(* PLC project common, CODESYS STW CODESYS V3.5 SP11 - ESX-3CS *)
(* stored: creationDateTime 2026-05-19T11:31:35.1210252, version 0.1, modificationDateTime 2026-01-27T11:29:48, organization Isoloader *)

TYPE t_can_message : CANMessage;
END_TYPE

TYPE t_can_message_set : ARRAY[1..32] OF POINTER TO t_can_message;
END_TYPE

TYPE t_long_string : STRING(72);
END_TYPE

TYPE t_long_string_reference : REFERENCE TO t_long_string;
END_TYPE

TYPE t_medium_string : STRING(16);
END_TYPE

TYPE t_medium_string_reference : REFERENCE TO t_medium_string;
END_TYPE

TYPE t_mediumlong_string : STRING(32);
END_TYPE

TYPE t_mediumlong_string_reference : REFERENCE TO t_mediumlong_string;
END_TYPE

TYPE t_ms_time : TIME;
END_TYPE

TYPE t_onoff_state : (cOnOffStateOff := 0, cOnOffStateTurningOn := 1, cOnOffStateOn := 2, cOnOffStateTurningOff := 3);
END_TYPE

TYPE t_percentage : REAL;
END_TYPE

TYPE t_short_string : STRING(8);
END_TYPE

TYPE t_short_string_reference : REFERENCE TO t_short_string;
END_TYPE

TYPE t_time : TIME;
END_TYPE

TYPE t_timer : Timer;
END_TYPE

TYPE t_system_handler : SystemHandler;
END_TYPE

VAR_GLOBAL CONSTANT  (* GlobalVariablesCommon *)
  cPi : REAL := 3.141592654;
  c2Pi : REAL := 6.283185307;
  cPiNegative : REAL := -3.141592654;
  cPIOn2 : REAL := 1.5708;
  cRelayCoilCurrentMinThreshold : WORD := 200;
  cRelayCoilCurrentMaxThreshold : WORD := 500;
  cRelayCoilResistanceThreshold : WORD := 80;
  cRelayCoilCurrentThreshold : WORD := 200;
  cRelayCoilTimeout : t_time := TIME#500ms;
  cRelayCoilTimeoutIndirect : t_time := TIME#600ms;
  gCodeErrorHandler : t_system_handler;
  gConfigErrorHandler : t_system_handler;
  gManualTemporaryOveride : BOOL := FALSE;
END_VAR

FUNCTION_BLOCK CANMessage
  VAR
    lSuccess : BOOL;
    lProceed : BOOL;
    lFinished : BOOL;
    lStarted : BOOL;
    lMessageCount : UINT := 0;
    lPostTimer : t_timer;
  END_VAR

            
          

METHOD finish
                  reset();

lStarted := TRUE;
lMessageCount := lMessageCount + 1;
                
END_METHOD

METHOD initialize
                  reset();

lMessageCount := 0;

lPostTimer.Enable := TRUE;
lPostTimer.Period := T#5S;
lPostTimer.initialize();
                
END_METHOD

METHOD operator
                  IF (NOT(Finished)) then
	lPostTimer.reset();
END_IF

lPostTimer.operator();

                
END_METHOD

METHOD reset
                  lSuccess := FALSE;
lProceed := FALSE;
lFinished := FALSE;
lStarted := FALSE;

                
END_METHOD

METHOD start
                  reset();

lStarted := TRUE;
lMessageCount := lMessageCount + 1;
                
END_METHOD

PROPERTY Finished : BOOL
GET
                    Finished := lFinished;
                  
END_GET
END_PROPERTY

PROPERTY PostPeriod : t_time
GET
                    PostPeriod := lPostTImer.Period;
                  
END_GET
SET
                    lPostTimer.Period := PostPeriod;
                  
END_SET
END_PROPERTY

PROPERTY Proceed : BOOL
GET
                    Proceed := lProceed;
                  
END_GET
END_PROPERTY

PROPERTY Running : BOOL
GET
                    Running := ((lStarted) and (NOT(lPostTimer.Expired)));
                  
END_GET
END_PROPERTY

PROPERTY Started : BOOL
GET
                    Started := lStarted;
                  
END_GET
END_PROPERTY

PROPERTY Success : BOOL
GET
                    Success := lSuccess;
                  
END_GET
END_PROPERTY
END_FUNCTION_BLOCK

FUNCTION_BLOCK CANMessageSequence EXTENDS CANMessage
  VAR
    lSequence : t_can_message_set;
    lSequenceCount : USINT := 0;
    lSequenceIndex : USINT := 0;
  END_VAR

            
          

METHOD initialize
  VAR
    i : USINT;
  END_VAR
                  SUPER^.initialize();

FOR i:=1 TO lSequenceCount DO
	lSequence[i]^.initialize();
END_FOR

                
END_METHOD

METHOD operator
  VAR
    b : BOOL;
  END_VAR
                  IF ((NOT(Enabled)) OR (NOT(Running))) THEN
	RETURN;
END_IF

SUPER^.operator();

lSequence[lSequenceIndex]^.operator();

IF (lSequence[lSequenceIndex]^.Finished) THEN
	IF (lSequence[lSequenceIndex]^.Proceed) THEN
		b:= lSequence[lSequenceIndex]^.Success;
		
		lSequenceIndex := lSequenceIndex + 1;
		IF (lSequenceIndex>lSequenceCount) THEN
			lSuccess := b;
			lFinished := TRUE;
			finish();
		ELSE
			lSequence[lSequenceIndex]^.start();	
		END_IF
	ELSE
		lSuccess := FALSE;
		lFinished := TRUE;
		finish();
	END_IF
END_IF

                
END_METHOD

METHOD registerMessage : POINTER TO t_can_message
  VAR_INPUT
    message : POINTER TO t_can_message;
  END_VAR
                  IF (lSequenceCount>32) THEN
	registerMessage := 0;
	RETURN;
END_IF

lSequenceCount := lSequenceCount + 1;
lSequence[lSequenceCount] := message;
                
END_METHOD

METHOD reset
  VAR
    i : USINT;
  END_VAR
                  SUPER^.reset();

lSequenceIndex := 0;

FOR i:=1 TO lSequenceCount DO
	lSequence[i]^.reset();
END_FOR


                
END_METHOD

METHOD start
                  SUPER^.reset();

IF (lSequenceCount=0) THEN
	lSequenceIndex := 0;
	RETURN;
END_IF

lSequenceIndex := 1;

lSequence[lSequenceIndex]^.start();

                
END_METHOD

PROPERTY Enabled : BOOL
GET
                    Enabled := (lSequenceIndex>0);

                  
END_GET
END_PROPERTY
END_FUNCTION_BLOCK

FUNCTION_BLOCK SystemHandler
  VAR_INPUT
    pResult : BYTE;
    pMessage : STRING;
    pFlag : BOOL;
  END_VAR
  VAR
    lState : BOOL := FALSE;
  END_VAR

            lState := TRUE;
          

METHOD reset
                  lState := FALSE;
                
END_METHOD
END_FUNCTION_BLOCK

FUNCTION_BLOCK Counter
  VAR
    lCount : USINT;
    lCountPrev : USINT;
    _Unique : UINT;
    lUnique : REFERENCE TO UINT := _Unique;
    lRising : BOOL;
    lFalling : BOOL;
    lHigh : BOOL;
  END_VAR

            
          

METHOD register
                  lCount := lCount + 1;
                
END_METHOD

METHOD operator
                  lRising := (lCountPrev=0) AND (lCount>0);
lFalling := (lCountPrev>0) AND (lCount=0);
lHigh := (lCount>0);

IF (lRising) THEN
	lUnique := lUnique + 1;
END_IF

lCountPrev := lCount;
lCount := 0;
                
END_METHOD

METHOD initialize
                  lCount := lCountPrev := 0;
lUnique := 0;
lRising := lFalling := lHigh := FALSE;
                
END_METHOD

METHOD reset
                  lCount := lCountPrev := 0;
lUnique := 0;
lRising := lFalling := lHigh := FALSE;

                
END_METHOD

METHOD setReference
  VAR_INPUT
    u : REFERENCE TO UINT;
  END_VAR
                  lUnique REF= u;
                
END_METHOD

PROPERTY Count : USINT
GET
                    Count := lCount;
                  
END_GET
END_PROPERTY

PROPERTY Rising : BOOL
GET
                    Rising := lRising;
                  
END_GET
END_PROPERTY

PROPERTY Falling : BOOL
GET
                    Falling := lFalling;
                  
END_GET
END_PROPERTY

PROPERTY High : BOOL
GET
                    High := lHigh;
                  
END_GET
END_PROPERTY

PROPERTY Unique : UINT
GET
                    Unique := lUnique;
                  
END_GET
END_PROPERTY
END_FUNCTION_BLOCK

FUNCTION strcmp : BOOL
  VAR_INPUT
    str1 : STRING;
    str2 : STRING;
  END_VAR
  VAR
    i : UINT;
    lng : UINT;
  END_VAR

            lng :=INT_TO_UINT(LEN(str1));

IF (lng<>INT_TO_UINT(LEN(str2))) THEN
	strcmp := FALSE;
	RETURN;
END_IF

FOR i:=0 TO lng DO
	IF (str1[i]<>str2[i]) THEN
		strcmp := FALSE;
		RETURN;
	END_IF
END_FOR

strcmp := TRUE;

          
END_FUNCTION

FUNCTION_BLOCK Timer
  VAR_INPUT
    lEnable : BOOL := FALSE;
    lPeriod : t_ms_time;
  END_VAR
  VAR
    lTimer : TON;
    lExpired : BOOL := FALSE;
  END_VAR

            ;
          

METHOD initialize
                  lExpired := FALSE;
                
END_METHOD

METHOD operator
                  lTimer(IN:=lEnable,PT:=lPeriod,Q=>lExpired);
                
END_METHOD

METHOD reset
                  lTimer(IN:=FALSE,PT:=lPeriod);
lExpired := FALSE;
                
END_METHOD

PROPERTY Enable : BOOL
GET
                    Enable := lEnable;
                  
END_GET
SET
                    lEnable := Enable;
                  
END_SET
END_PROPERTY

PROPERTY Expired : BOOL
GET
                    Expired := lExpired;
                  
END_GET
END_PROPERTY

PROPERTY Period : t_time
GET
                    Period := lPeriod;
                  
END_GET
SET
                    lPeriod := Period;
                  
END_SET
END_PROPERTY
END_FUNCTION_BLOCK

FUNCTION_BLOCK TimerWithStatistics EXTENDS Timer
  VAR
    lUnexpiredMax : t_time := TIME#0ms;
  END_VAR

            
          

METHOD reset
                  IF (NOT(lExpired)) THEN
	lUnexpiredMax := MAX(lUnexpiredMax,lTimer.ET);
END_IF

SUPER^.reset();

                
END_METHOD

PROPERTY UnexpiredMax : t_time
GET
                    UnexpiredMax := lUnexpiredMax;
                  
END_GET
END_PROPERTY
END_FUNCTION_BLOCK
